PROGRAM MAIN
VAR
	hydValve : HydraulicValve();
	monError	:	Monitoring_Error();
	enaNegDirB : BOOL := FALSE;
	enaPosDirB : BOOL := FALSE;
	commandSet : REAL := 0;
	currentError	:	BOOL := FALSE;
	//konfiguraParametry : REFERENCE TO configaracionParammetrs  REF=generalVariable.conParammetr;
	OutPosDir : REAL := 0 ;	// Výstup v daném směru [mA]
	OutNegDir : REAL := 0 ;	// Výstup v daném směru [mA]
END_VAR

// control whether the valve is in operation, whether it is possible to enter a new value and  direction command
IF NOT(generalVariable.staus.bBussy) THEN 
	monError(negDirB := enaNegDirB, posDirB := enaPosDirB, command := commandSet);
	IF NOT(monError.currentError) THEN
		hydValve(bvNegDir := enaNegDirB, bvPosDir := enaPosDirB, command := commandSet); 
	END_IF
END_IF
OutPosDir := convertToAm(generalVariable.staus.OutPosDirProc * 10, TRUE);
OutNegDir := convertToAm(generalVariable.staus.OutNegDirProc * 10, FALSE);

END_PROGRAM

(* stored: Version 1.1.0.1, ProductVersion 3.1.4024.12
   POU MAIN: Id {4d8a33a6-50bf-43f1-9baa-ca9df7252f1c}, SpecialFunc None *)
